// TIA Portal V20 export
TYPE "UDT_PartStates"
   STRUCT
      BW : Struct
         Good : Bool;
         Unknown : Bool;
         Bad : Bool;
         Absent : Bool;
         PresentUnexpected : Bool;
         AbsentUnexpected : Bool;
      END_STRUCT;
      Part : Struct
         Good : Bool;
         Unknown : Bool;
         Bad : Bool;
         Absent : Bool;
         PresentUnexpected : Bool;
         AbsentUnexpected : Bool;
      END_STRUCT;
   END_STRUCT;
END_TYPE
